(* Logix 5000 project; controller Lab2_Unit18 vendor 1 type 14 code 106 rev 30.11; software revision 30.00 *)

TASK MainTask (continuous, watchdog 500 ms) : MainProgram

MODULES
   Local : vendor 1 type 14 code 106 (Compact 0, rev 30.11)
      I1 : 1769-IQ16 (Compact 1, rev 1.1, Input RPI 20 ms)
      A3 : vendor 1 type 10 code 33 (Compact 3, rev 1.1, Output RPI 80 ms)
      O2 : vendor 1 type 7 code 86 (Compact 2, rev 2.1, Output RPI 20 ms)
END_MODULES

PROGRAM MainProgram   (* main routine MainRoutine *)

ROUTINE MainRoutine   (* ladder *)
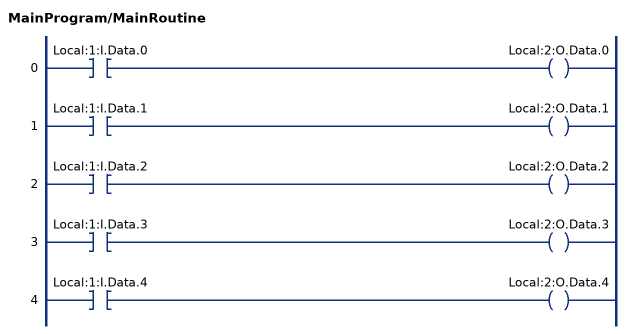
   0: XIC(Local:1:I.Data.0)OTE(Local:2:O.Data.0);
   1: XIC(Local:1:I.Data.1)OTE(Local:2:O.Data.1);
   2: XIC(Local:1:I.Data.2)OTE(Local:2:O.Data.2);
   3: XIC(Local:1:I.Data.3)OTE(Local:2:O.Data.3);
   4: XIC(Local:1:I.Data.4)OTE(Local:2:O.Data.4);
END_ROUTINE
END_PROGRAM
